FUNCTION_BLOCK ACCESS_DB
  {SET_ATTRIBUTE(OpcUa, SERVICE)}
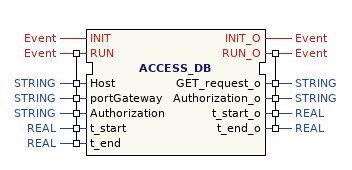
  EVENT_INPUT
    INIT;
    RUN WITH Host, portGateway, Authorization, t_start, t_end; {SET_ATTRIBUTE(OpcUa, Method)}
  END_EVENT
  EVENT_OUTPUT
    INIT_O;
    RUN_O WITH GET_request_o, Authorization_o, t_start_o, t_end_o;
  END_EVENT
  VAR_INPUT
    Host : STRING; {SET_ATTRIBUTE(OpcUa, Variable.RUN)}
    portGateway : STRING; {SET_ATTRIBUTE(OpcUa, Variable.RUN)}
    Authorization : STRING; {SET_ATTRIBUTE(OpcUa, Variable.RUN)}
    t_start : REAL; {SET_ATTRIBUTE(OpcUa, Variable.RUN)}
    t_end : REAL; {SET_ATTRIBUTE(OpcUa, Variable.RUN)}
  END_VAR
  VAR_OUTPUT
    GET_request_o : STRING; {SET_ATTRIBUTE(OpcUa, Variable.RUN)}
    Authorization_o : STRING; {SET_ATTRIBUTE(OpcUa, Variable.RUN)}
    t_start_o : REAL; {SET_ATTRIBUTE(OpcUa, Variable.RUN)}
    t_end_o : REAL; {SET_ATTRIBUTE(OpcUa, Variable.RUN)}
  END_VAR
END_FUNCTION_BLOCK
